// TIA Portal V16 export
// export: Created 2021-08-16T20:43:24.047403Z, ExportSetting WithDefaults, DisplayName Totally Integrated Automation Portal, DisplayVersion V16, DisplayName TIA Portal Version Control Interface, DisplayVersion V16, DisplayName TIA Portal Openness, DisplayVersion V16, DisplayName STEP 7 Professional, DisplayVersion V16, DisplayName STEP 7 Safety, DisplayVersion V16, DisplayName WinCC Advanced, DisplayVersion V16
VAR_GLOBAL   // PLC tag table "Input & Output table"
   "Conveyor 1" AT %Q0.0 : Bool;
   "Conveyor 2" AT %Q0.1 : Bool;
   Green AT %Q0.2 : Bool;
   Yellow AT %Q0.3 : Bool;
   Red AT %Q0.4 : Bool;
END_VAR
